{attribute 'qualified_only'}
VAR_GLOBAL
	
	//OPMODE_CSP : SINT := 8;
	OPMODE_CSV : SINT := 9;
	OPMODE_CST : SINT := 10;
	
	OPMODE_STRINGS : ARRAY [1..2] OF STRING := ['CSV', 'CST']; 
	
	TARGET_AMPLITUDE : DINT := 100;
	SINUS_FREQUENCY : TIME := T#300MS; // Milliseconds
	AMPLITUDE_OFFSET : REAL := 0.0;

	
	RESET_HOLD_TIME : TIME := T#2S; // Reset time
	RESET_SIGNAL : TIME := T#10S; // Cycle time (Checks after n seconds for errors)

	velocity_in AT %I*:DINT;
	velocity_out AT %Q*: DINT;
	torque_out AT %Q*: INT;
	opmode AT %Q*: SINT := OPMODE_CST;
	
	NET_ID_CABINET : T_AmsNetID := '192.168.101.251.3.1';
	SLAVE_ADDR : UINT := 1001;
	OBJ_DIR_ERROR			: WORD := 16#203F;
	NO_ERROR : LINT := 16#20746C7561466F4E;
	STR_NO_ERROR : STRING := LINT_TO_STRING(NO_ERROR);
END_VAR

(* stored: Version 1.1.0.1, ProductVersion 3.1.4022.18
   GVL GVL: Id {99f84099-7a89-4751-976f-dd68e9193fbb} *)
